// TwinCAT 3 PLC project PLC
// ProgramVersion: 3.1.4026.20
// CompilerDefines: VISU_USEPROPERTYINFO
// libraries:
//   Tc2_MC2, * (Beckhoff Automation GmbH)
//   Tc2_Standard, * (Beckhoff Automation GmbH)
//   Tc2_System, * (Beckhoff Automation GmbH)
// project tree:
//   DUTs/ enum_states.TcDUT
//   / GlobalTextList.TcGTLO, PlcTask.TcTTO, Visualization Manager.TcVMO (not stored)
//   GVLs/ IFC_HW.TcGVL (not stored)
//   POUs/Fehlerbehandlung/ FB_TimeOutError.TcPOU
//   POUs/HardwareEbene/ FB_CNV.TcPOU
//   POUs/ MAIN.TcPOU
//   POUs/ModulEbene/ FB_Transportband.TcPOU
//   POUs/ProzessEbene/ FB_Vereinzelung.TcPOU
//   POUs/Utility/ FB_Blink.TcPOU, FB_DigitalInput.TcPOU
// (motion and I/O tree: see PLC project tempmodel)
// real-time tasks:
//   TASK PlcTask: cycle T#10ms, priority 21, ADS port 350
//   TASK PlcTask1: cycle T#10ms, priority 22, ADS port 351
//   TASK PlcTask2: cycle T#10ms, priority 20, ADS port 352
// variable links:
//   LF_System_PLC/LF_System_PLC Instance <-> PLC/PLC Instance
//     PlcTask Inputs/MAIN.bIn_LedRot <-> PlcTask Outputs/IFC_HW.bAmpelRot
//   PLC/PLC Instance <-> NC-Task 1 SAF/Axes/BandAchse
//     PlcTask Inputs/IFC_HW.ax_BandMotor.NcToPlc <-> Outputs/ToPlc
//     PlcTask Outputs/IFC_HW.ax_BandMotor.PlcToNc <-> Inputs/FromPlc

CONFIGURATION PLC
    RESOURCE PLC ON TwinCAT3
        TASK PlcTask(INTERVAL := T#10ms, PRIORITY := 20);
        PROGRAM MAIN WITH PlcTask : MAIN;
    END_RESOURCE
END_CONFIGURATION

// ---- DUTs/enum_states.TcDUT
{attribute 'qualified_only'}
{attribute 'strict'}
{attribute 'to_string'}
TYPE enum_states :
(
	error, // rot blinken
	stop, // Rot, Gelb blinkem
	off, // Rot leuchten
	init, // Grün blinken
	production, // grün leuchten
	ready, // gelb, grün blinken
	done, // geld, grün leuchten
	setup // gelb blinken
);
END_TYPE

// ---- POUs/MAIN.TcPOU
PROGRAM MAIN
VAR
	fb_Vereinzelung : FB_Vereinzelung;
	fb_CNV : FB_CNV; 
	bSens1: BOOL;
	bSens2: BOOL;
	bSens3: BOOL;
	fbEndXmin : FB_DigitalInput(TRUE);
	
	bError : BOOL;
	ErrorID : DWORD;
	reset : BOOL;
END_VAR

fb_Vereinzelung(
	bEnable:= IFC_HW.bEnable, 
	bExecute:= IFC_HW.bExecute, 
	bSens1:= IFC_HW.bEinzelSens3, //Achtung hab ich vertauscht
	bSens2:= IFC_HW.bEinzelSens2, 
	bSens3:= IFC_HW.bEinzelSens1); //Achtung hab ich vertauscht 
	
// Schleuse oben
IF fb_Vereinzelung.bGate1 THEN 
    IFC_HW.bR1AKT1 := TRUE;   // oben öffnen
    IFC_HW.bR2AKT1 := FALSE;  // oben schließen aus
ELSE 
    IFC_HW.bR1AKT1 := FALSE;  
    IFC_HW.bR2AKT1 := TRUE;   // oben schließen
END_IF;

// Schleuse unten
IF fb_Vereinzelung.bGate2 THEN
    IFC_HW.bR1AKT2 := TRUE;   // unten öffnen
    IFC_HW.bR2AKT2 := FALSE;  // unten schließen aus
ELSE
    IFC_HW.bR1AKT2 := FALSE;
    IFC_HW.bR2AKT2 := TRUE;   // unten schließen
END_IF;

fb_CNV(
	bEnable:= IFC_HW.bEnable, 
	bExecute:= IFC_HW.bExecute, 
	bHalt:= IFC_HW.bBandSens1, 
	rVel:= 500, 
	//eState=> , 
	ax:= IFC_HW.ax_BandMotor);
	
fbEndXmin(bSensSignal:= Ifc_HW.bManEndXmin, bSensLogic=> );

// zum Wert auslesen
IF fbEndXmin.bSensLogic THEN
	// Achse dadrf nciht in negative Richtung fahren
END_IF

// in der main das instanzieren
// fbAbfuellmodul instanzieren
// 	bEnable := ifc_hw.bEnable ,
// 	bExecute := ifc_hw.bExecute,
// bStop := ,
// 

// das hier bleibt in der main
IF bError AND (ErrorID = 9001 OR ErrorID = 9003) THEN
	ifc_hw.bStop := TRUE;
END_IF



ifc_hw.bereset := reset;

IF bError AND reset THEN
	ifc_hw.bStop := FALSE;
	reset := FALSE;
END_IF

// im ifc eine globale vairable schreiben breset

END_PROGRAM

// ---- POUs/ProzessEbene/FB_Vereinzelung.TcPOU
FUNCTION_BLOCK FB_Vereinzelung
VAR_INPUT
	
	bEnable : BOOL; //Bedienereingabe
	bExecute: BOOL; //Bedienereingabe 
	
	bSens1 : BOOL; //Flasche in Kamnmer
	bSens2 : BOOL; // Flasche in Speicher 
	bSens3 : BOOL; //Flasche am Kopf
	
END_VAR

VAR_OUTPUT
	bGate1 : BOOL; //Schleuse oben, wenn TRUE = Öffnen
	bGate2: BOOL; //Schleuse unten, wenn TRUE = Öffnen 
	nState : INT; //Variable für die CASE-Anweisung
END_VAR
VAR
	tClose : TON; //Timer zum Schließen 
	tCloseTime : TIME := T#1000MS; 
END_VAR

IF NOT bEnable OR NOT bExecute THEN 
	bGate1 := FALSE; 
	bGate2 := FALSE;
	nState := 0; //Zustand auf IDLE bzw. ausgangslage setzen 
	tClose(IN := FALSE, PT := tCloseTime);

ELSE 
	CASE nState OF 
		0: //Warten auf Start mit bEnable und bExecute 
			bGate1 := FALSE; 
			bGate2 := FALSE; 
			tClose(IN := FALSE, PT := tCloseTime);
			
			IF bExecute THEN 
				nState := 1; //Wenn Execute dann auf State 1 Wechseln
			END_IF
		
		1: //Warten auf Flasche im Speicher 
			bGate1 := FALSE; 
			bGate2 := FALSE;
			tClose(IN := FALSE, PT := tCloseTime);
			
			IF bSens2 THEN 
				nState := 2; // Wenn Flasche in Speicher dann Zustand 2
			END_IF
		
		2: //obere Schleuse öffnen 
			bGate1 := TRUE; //Obere Schleuse wird geöffnet 
			bGate2 := FALSE; 
			tClose(IN := FALSE, PT := tCloseTime);
			
			IF bSens1 THEN 
				nState := 3; // Wenn Flasche in Kammer dann zu Zustand 3
			END_IF
		3: //obere Schleuse schließen 
			bGate1 := FALSE; 
			bGate2 := FALSE;
			tClose(IN := TRUE, PT := tCloseTime); // Zeit zum schließen
			
			IF tClose.Q THEN //Wenn geschlossen zurücksetzen und Zustand 4 wechseln
				tClose(IN := FALSE, PT := tCloseTime);
				nState := 4;
			END_IF
		4: //Untere Schleuse öffnen 
			bGate1 := FALSE;
			bGate2 := TRUE; //untere schleuse wird geöffnet
			tClose(IN := FALSE, PT := tCloseTime);
			
			IF NOT bSens1 THEN 
				nState := 5;
			END_IF
		5: // Untere Schleuse Schließen
			bGate1 := FALSE;
			bGate2 := FALSE; //untere schleuse wird geschlossen
			tClose(IN := TRUE, PT := tCloseTime);
			
			IF tClose.Q THEN 
				tClose(IN := FALSE, PT := tCloseTime);
				nState := 1;
			END_IF
			
		ELSE //Falls irgend was anderes eintritt zustand 0 
			bGate1 := FALSE; 
			bGate2 := FALSE; 
			tClose(IN := FALSE, PT := tCLoseTime);
			nState := 0; 
	END_CASE
END_IF

END_FUNCTION_BLOCK

// ---- POUs/HardwareEbene/FB_CNV.TcPOU
FUNCTION_BLOCK FB_CNV
VAR_INPUT
	// Steuereingänge
	bEnable : BOOL;
	bExecute : BOOL;
	bHalt : BOOL;
	
	// Bewegungseigenschaften
	rVel : REAL;
END_VAR
VAR_OUTPUT
	//eState : E_State; // bzw je nachdem wie meine enumeration genannt ist
END_VAR
VAR
	nState : INT := 0;
	mcPower : MC_Power;
	mcReset : MC_Reset;
	mcVelocity : MC_MoveVelocity;
	mcHalt : MC_Halt;
	bStop : BOOL;
	mcStop : MC_Stop;
END_VAR

// für achsenreferenz neue Variablen bereich
VAR_IN_OUT
	ax : Axis_Ref;
END_VAR

mcPower(
	Axis:= ax, 
	Enable:= , 
	Enable_Positive:= , 
	Enable_Negative:= , 
	Override:= , 
	BufferMode:= , 
	Options:= , 
	Status=> , 
	Busy=> , 
	Error=> , 
	ErrorID=> );
	
mcReset(
	Axis:= ax, 
	Execute:= , 
	Done=> , 
	Busy=> , 
	Error=> , 
	ErrorID=> );
	
mcVelocity(
	Axis:= ax, 
	Execute:= , 
	Velocity:= rVel, 
	Acceleration:= , 
	Deceleration:= , 
	Jerk:= , 
	Direction:= , 
	BufferMode:= , 
	Options:= , 
	InVelocity=> , 
	Busy=> , 
	Active=> , 
	CommandAborted=> , 
	Error=> , 
	ErrorID=> );
	
mcHalt(
	Axis:= ax, 
	Execute:= , 
	Deceleration:= , 
	Jerk:= , 
	BufferMode:= , 
	Options:= , 
	Done=> , 
	Busy=> , 
	Active=> , 
	CommandAborted=> , 
	Error=> , 
	ErrorID=> );

ax.ReadStatus(); // info der Achse zyklisch holen

bStop := ifc_Hw.bStop;

IF bStop THEN
	nState = 80; // Stop conveyer
	
END_IF

IF ax.Status.Error THEN
	nState := 99; // Error State

ELSIF NOT bEnable THEN
	nState := 0; // Off
END_IF

CASE nState OF
	0: // Off
	mcPower.Enable := FALSE;
	mcPower.Enable_Positive := FALSE;
	mcReset.Execute := FALSE;
	mcVelocity.Execute := FALSE;
	mcHalt.Execute := FALSE;
	
	
	IF ax.Status.Error THEN
		nState := 99; // Error State
	ELSIF bEnable THEN
		nState := 1; // INIT
	END_IF
	
	1: // Init
	mcPower.Enable := TRUE;
	mcPower.Enable_Positive := TRUE;
	mcReset.Execute := FALSE;
	mcVelocity.Execute := FALSE;
	mcHalt.Execute := FALSE;
	
	IF mcPower.Status THEN
		nState := 2; // READY
	END_IF
	
	2: // Ready
	mcPower.Enable := TRUE;
	mcPower.Enable_Positive := TRUE;
	mcReset.Execute := FALSE;
	mcVelocity.Execute := FALSE;
	mcHalt.Execute := FALSE;
	
	IF bExecute THEN
		nState := 3; // CNV an
	END_IF
	
	3: // CNV an
	mcPower.Enable := TRUE;
	mcPower.Enable_Positive := TRUE;
	mcReset.Execute := FALSE;
	mcVelocity.Execute := TRUE;
	mcHalt.Execute := FALSE;
	
	IF bHalt THEN
		nState := 4; // CNV aus
	END_IF
	
	4: // CNV aus
	mcPower.Enable := TRUE;
	mcPower.Enable_Positive := TRUE;
	mcReset.Execute := FALSE;
	mcVelocity.Execute := FALSE;
	mcHalt.Execute := TRUE;
	
	IF mcHalt.Done THEN
		nState := 5; // DONE
	END_IF
	
	5: // Done (Stillstand nach Bewegung)
	mcPower.Enable := TRUE;
	mcPower.Enable_Positive := TRUE;
	mcReset.Execute := FALSE;
	mcVelocity.Execute := FALSE;
	mcHalt.Execute := FALSE;
	
	IF NOT bExecute AND NOT bHalt THEN
		nState := 2; // READY 
	END_IF
	
	80: // Stop cNV
	mcVelocity.Execute := FALSE;
	mcHalt.Execute := FALSE;
	mcStop.Execute := TRUE;
	
	IF mcStop.Done AND NOT bStop THEN
		nState := 81;
	END_IF
	
	81: // Re-Init
	mcVelocity.Execute := FALSE;
	mcHalt.Execute := FALSE;
	mcStop.Execute := FALSE;
	mcReset.Execute := TRUE;
	
	IF mcReset.Done THEN
		nState := 3;
	END_IF
	
	
	99: // Error State
	mcPower.Enable := FALSE;
	mcPower.Enable_Positive := FALSE;
	mcReset.Execute := FALSE;
	mcVelocity.Execute := FALSE;
	mcHalt.Execute := FALSE;
	
	IF bEnable THEN
		nState := 100; // Resolve
	END_IF
	
	100: // Resolve
	mcPower.Enable := FALSE;
	mcPower.Enable_Positive := FALSE;
	mcReset.Execute := TRUE;
	mcVelocity.Execute := FALSE;
	mcHalt.Execute := FALSE;
	
	IF mcReset.Done THEN
		nState := 1; // Init
	END_IF
	
END_CASE

END_FUNCTION_BLOCK

// ---- POUs/Utility/FB_DigitalInput.TcPOU
FUNCTION_BLOCK FB_DigitalInput
VAR_INPUT
	bSensSignal : BOOL;
END_VAR
VAR_OUTPUT
	bSensLogic : BOOL; 
END_VAR
VAR
	_Invert : BOOL := FALSE;
END_VAR

IF _Invert THEN
	bSensLogic := NOT bSensSignal;
ELSE	
	bSensLogic := bSensSignal;
END_IF

//FB_Init is always available implicitly and it is used primarily for initialization.
//The return value is not evaluated. For a specific influence, you can also declare the
//methods explicitly and provide additional code there with the standard initialization
//code. You can evaluate the return value.
METHOD FB_Init: BOOL
VAR_INPUT
    bInitRetains: BOOL; // TRUE: the retain variables are initialized (reset warm / reset cold)
    bInCopyCode: BOOL;  // TRUE: the instance will be copied to the copy code afterward (online change)   
	Invert : BOOL;
END_VAR
_Invert := Invert;
END_METHOD

END_FUNCTION_BLOCK

// ---- POUs/Fehlerbehandlung/FB_TimeOutError.TcPOU
FUNCTION_BLOCK FB_TimeOutError
VAR_INPUT // siehe handy bild für rest
	bReset : BOOL;
	bIN : BOOL;
	bZiel : BOOL;
END_VAR
VAR_OUTPUT
	bError : BOOL;
	ErrorID : BOOL;
END_VAR
VAR
	timer : Ton;
END_VAR

// FB_transport
// fehlerdirektionsbausteine
//fbTO _Transport : FB_TimeOutError(9001, T#10S);
// ausgänge erweitern
//bError : BOOL;
//ErrorID : DWORD;
// rbtO_Transport : FB_timeouterror(9001, T#10s);
// in die normale VAR
bStop : BOOL;


// im prgrammteil instanzieren
fbTO_TransportTHIS^(
	bReset:= , 
	bIN:= eState = E_Satet.Produtction, 
	bZiel:= eState = E_State.Done, 
	bError=> bError, 
	ErrorID=> ErrorID);

bStop := ifc_hw.bStop;
// dann um die Case of eine If machen wo wir bStop abfragen

// FB Filling modul 
// im tunktionsaufruf der fbtransport
// ausgänge erweitern
// bError : BOOL;
// ErrorID : DWORD;
// nMemState : INT;

// variable für bStop anlegen
bStop : BOOL;
// programmblock
bStop := ifc_hw.bStop;
IF bStop THEN
	nMemState := nState;
END_IF



timer(IN:= , PT:=_PT, Q=> , ET=> );

IF bIN THEN
	timer.In := TRUE;
END_IF

IF bZiel THEN
	timer.IN := FALSE;
END_IF

IF timer.Q THEN
	bError := TRUE;
	ErrorID := _ErrorID;
ELSIF NOT timer.Q OR bReset THEN
	bError := FALSE;
	ErrorID := 0;

//FB_Init is always available implicitly and it is used primarily for initialization.
//The return value is not evaluated. For a specific influence, you can also declare the
//methods explicitly and provide additional code there with the standard initialization
//code. You can evaluate the return value.
METHOD FB_Init: BOOL
VAR_INPUT
    bInitRetains: BOOL; // TRUE: the retain variables are initialized (reset warm / reset cold)
    bInCopyCode: BOOL;  // TRUE: the instance will be copied to the copy code afterward (online change)
	ErrorID : DWORD;
	PT : Time;   
END_VAR
_ErrorID := ErrorID; 
_PT := PT;
END_METHOD

END_FUNCTION_BLOCK

// ---- POUs/ModulEbene/FB_Transportband.TcPOU
FUNCTION_BLOCK FB_AbfuellModul
VAR_INPUT
	bEnable : BOOL;
	bExecute : BOOL;
END_VAR
VAR_OUTPUT
	eState : BOOL;
END_VAR
VAR
	FB_Transport : BOOL;
	FB_Vereinzelung : BOOL;
	FB_Disp : BOOL;
	nState : INT;
	nStation : INT := 0; // bei welcher Station wir aktuell sind, dann wird +1 gezhält
END_VAR

// Startzustand
IF NOT bEnable OR NOT bExecute THEN
	nState := 0;

ELSE
	
	CASE nState OF 
		0: // OFF
		bEnable := FALSE;
		bExecute := FALSE;
		FB_CNV.bEnable := FALSE;
		FB_CNV.bExecute := FALSE;
		FB_CNV.bHalt := FALSE;
		
		IF bEnable THEN
			nState := 1; // wenn bEnable gehen wir in 2. Case rein
		END_IF
		
		1: // Init
		bEnable := FALSE;
		bExecute := FALSE;
		FB_CNV.bEnable := TRUE;
		FB_CNV.bExecute := FALSE;
		FB_CNV.bHalt := FALSE;
		
		2: // Ready
		
		
	END_CASE



END_IF

END_FUNCTION_BLOCK

// ---- POUs/Utility/FB_Blink.TcPOU
FUNCTION_BLOCK FB_Blink
// Enumerationen einbinden mit den Zuständen
VAR_INPUT
   	State : enum_states;
END_VAR

VAR_OUTPUT
	
	// Output Signale für Ampel
	//bAmpelRot : IFC_HW;			// Signal-LED Rot
	//bAmpelGelb : IFC_HW;			// Signal-LED Gelb
	//bAmpelGrun : IFC_HW;

	bAmpelRot : BOOL;			// Signal-LED Rot
	bAmpelGelb : BOOL;			// Signal-LED Gelb
	bAmpelGrun : BOOL;
END_VAR

VAR
	fbTon   : TON;
	bBlink  : BOOL;
END_VAR


bAmpelRot := FALSE;
bAmpelGelb := FALSE;
bAmpelGrun := FALSE;

// einfacher Blinkgenerator
fbTon(IN := NOT fbTon.Q, PT := T#500ms);
IF fbTon.Q THEN
    bBlink := NOT bBlink;
END_IF;

CASE State OF
    State.off:
        bAmpelRot := TRUE;

    State.init:
        bAmpelGrun := bBlink;

    State.ready:
        bAmpelGelb := bBlink;
        bAmpelGrun := bBlink;

    State.production:
        bAmpelGrun := TRUE;

    State.done:
        bAmpelGelb := TRUE;
        bAmpelGrun := TRUE;

    State.error:
        bAmpelRot := bBlink;

    State.stop:
        bAmpelRot := bBlink;
        bAmpelGelb := bBlink;

    State.setup:
        bAmpelGelb := bBlink;
END_CASE;

END_FUNCTION_BLOCK
